// TIA Portal V16 export
// export: Created 2024-04-26T21:24:40.8001835Z, ExportSetting WithDefaults, DisplayName Totally Integrated Automation Portal, DisplayVersion V16, DisplayName TIA Portal Version Control Interface, DisplayVersion V16, DisplayName TIA Portal Openness, DisplayVersion V16, DisplayName STEP 7 Professional, DisplayVersion V16, DisplayName STEP 7 Safety, DisplayVersion V16, DisplayName WinCC Professional, DisplayVersion V16
ORGANIZATION_BLOCK "Main"   // OB1, LAD, ProgramCycle
TITLE = "Main Program Sweep (Cycle)"
{ S7_Optimized_Access := 'TRUE' }
VERSION : 0.1
// stored: AutoNumber true, IsIECCheckEnabled false, SetENOAutomatically false
   VAR_INPUT
      Initial_Call : Bool;   // Initial call of this OB
      Remanence : Bool;   // =True, if remanent data are available
   END_VAR
   VAR CONSTANT
      pozycja : Real := 45.0;
   END_VAR
   VAR_TEMP   // added for the SCL form of the ladder/FBD networks
      _w1 : Bool;
      _w2 : Bool;
   END_VAR
BEGIN

REGION Network 1: załączenie osi
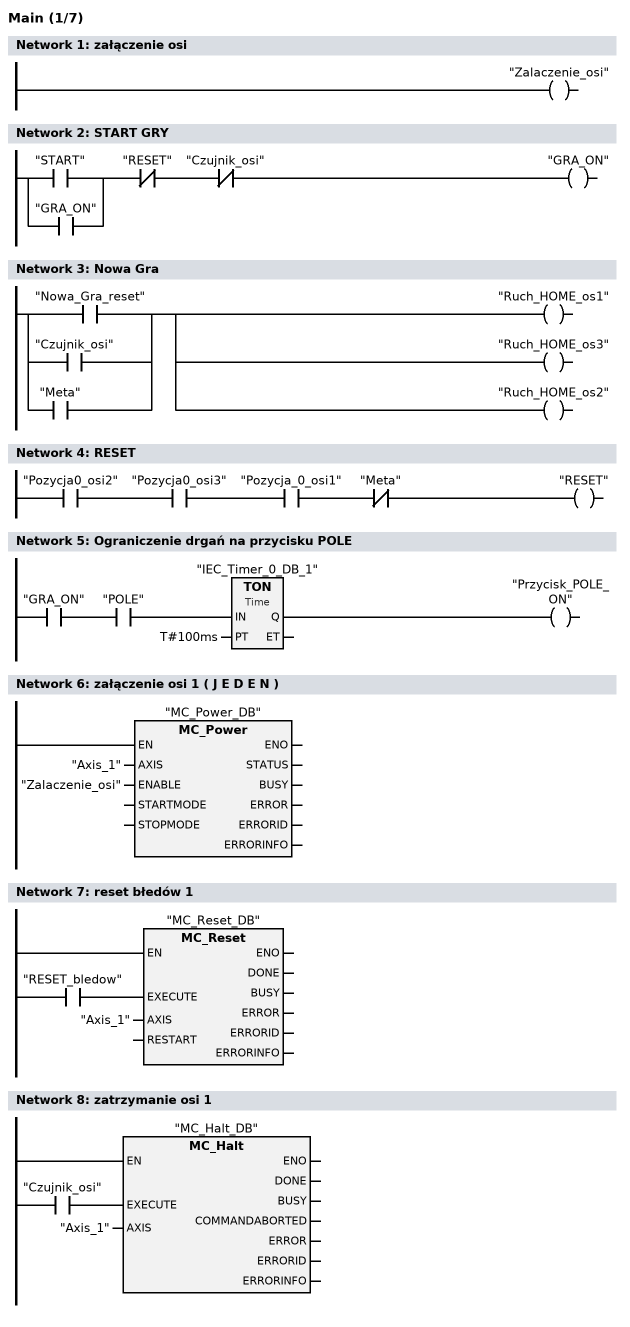
   RUNG wire#powerrail
      Coil( "Zalaczenie_osi" )
   END_RUNG
   // the same network as SCL:
   "Zalaczenie_osi" := TRUE;
END_REGION

REGION Network 2: START GRY
   RUNG wire#powerrail
      Contact( "START" )
      wire#w1
      I_Contact( "RESET" )
      I_Contact( "Czujnik_osi" )
      Coil( "GRA_ON" )
   END_RUNG
   RUNG wire#powerrail
      Contact( "GRA_ON" )
   END_RUNG wire#w1
   // the same network as SCL:
   "GRA_ON" := ("START" OR "GRA_ON") AND NOT "RESET" AND NOT "Czujnik_osi";
END_REGION

REGION Network 3: Nowa Gra
   RUNG wire#powerrail
      Contact( "Nowa_Gra_reset" )
      wire#w1
      Coil( "Ruch_HOME_os1" )
   END_RUNG
   RUNG wire#powerrail
      Contact( "Czujnik_osi" )
   END_RUNG wire#w1
   RUNG wire#powerrail
      Contact( "Meta" )
   END_RUNG wire#w1
   RUNG wire#w1
      Coil( "Ruch_HOME_os3" )
   END_RUNG
   RUNG wire#w1
      Coil( "Ruch_HOME_os2" )
   END_RUNG
   // the same network as SCL:
   "Ruch_HOME_os1" := "Nowa_Gra_reset" OR "Czujnik_osi" OR "Meta";
   "Ruch_HOME_os3" := "Ruch_HOME_os1";
   "Ruch_HOME_os2" := "Ruch_HOME_os1";
END_REGION

REGION Network 4: RESET
   RUNG wire#powerrail
      Contact( "Pozycja0_osi2" )
      Contact( "Pozycja0_osi3" )
      Contact( "Pozycja_0_osi1" )
      I_Contact( "Meta" )
      Coil( "RESET" )
   END_RUNG
   // the same network as SCL:
   "RESET" := "Pozycja0_osi2" AND "Pozycja0_osi3" AND "Pozycja_0_osi1" AND NOT "Meta";
END_REGION

REGION Network 5: Ograniczenie drgań na przycisku POLE
   RUNG wire#powerrail
      Contact( "GRA_ON" )
      Contact( "POLE" )
      { S7_Templates := "time_type := Time" } "IEC_Timer_0_DB_1".TON(pt := T#100ms, et =>)
      Coil( "Przycisk_POLE_ON" )
   END_RUNG
   // the same network as SCL:
   "IEC_Timer_0_DB_1".TON(IN := "GRA_ON" AND "POLE", PT := T#100ms);
   "Przycisk_POLE_ON" := "IEC_Timer_0_DB_1".Q;
END_REGION

REGION Network 6: załączenie osi 1 ( J E D E N )
   RUNG wire#powerrail
      "MC_Power_DB".MC_Power(Axis := "Axis_1", Enable := "Zalaczenie_osi", StartMode :=, StopMode :=, Status =>, Busy =>, Error =>, ErrorID =>, ErrorInfo =>)
   END_RUNG
   // the same network as SCL:
   "MC_Power_DB"(Axis := "Axis_1", Enable := "Zalaczenie_osi");   // MC_Power
END_REGION

REGION Network 7: reset błedów 1
   RUNG wire#powerrail
      "MC_Reset_DB".MC_Reset(Execute := wire#w1, Axis := "Axis_1", Restart :=, Done =>, Busy =>, Error =>, ErrorID =>, ErrorInfo =>)
   END_RUNG
   RUNG wire#powerrail
      Contact( "RESET_bledow" )
   END_RUNG wire#w1
   // the same network as SCL:
   "MC_Reset_DB"(Execute := "RESET_bledow", Axis := "Axis_1");   // MC_Reset
END_REGION

REGION Network 8: zatrzymanie osi 1
   RUNG wire#powerrail
      "MC_Halt_DB".MC_Halt(Execute := wire#w1, Axis := "Axis_1", Done =>, Busy =>, CommandAborted =>, Error =>, ErrorID =>, ErrorInfo =>)
   END_RUNG
   RUNG wire#powerrail
      Contact( "Czujnik_osi" )
   END_RUNG wire#w1
   // the same network as SCL:
   "MC_Halt_DB"(Execute := "Czujnik_osi", Axis := "Axis_1");   // MC_Halt
END_REGION

REGION Network 9: pozycjonowanie osi 1
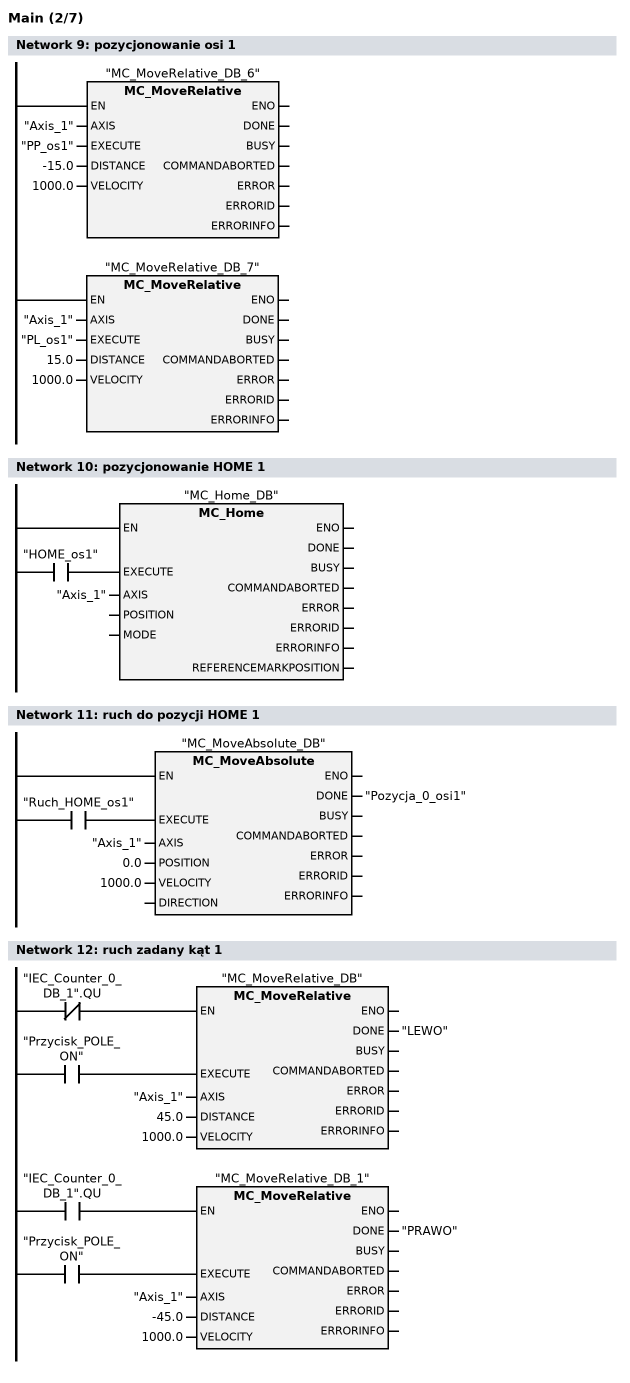
   RUNG wire#powerrail
      "MC_MoveRelative_DB_6".MC_MoveRelative(Axis := "Axis_1", Execute := "PP_os1", Distance := -15.0, Velocity := 1000.0, Done =>, Busy =>, CommandAborted =>, Error =>, ErrorID =>, ErrorInfo =>)
   END_RUNG
   RUNG wire#powerrail
      "MC_MoveRelative_DB_7".MC_MoveRelative(Axis := "Axis_1", Execute := "PL_os1", Distance := 15.0, Velocity := 1000.0, Done =>, Busy =>, CommandAborted =>, Error =>, ErrorID =>, ErrorInfo =>)
   END_RUNG
   // the same network as SCL:
   "MC_MoveRelative_DB_6"(Axis := "Axis_1", Execute := "PP_os1", Distance := -15.0, Velocity := 1000.0);   // MC_MoveRelative
   "MC_MoveRelative_DB_7"(Axis := "Axis_1", Execute := "PL_os1", Distance := 15.0, Velocity := 1000.0);   // MC_MoveRelative
END_REGION

REGION Network 10: pozycjonowanie HOME 1
   RUNG wire#powerrail
      "MC_Home_DB".MC_Home(Execute := wire#w1, Axis := "Axis_1", Position :=, Mode :=, Done =>, Busy =>, CommandAborted =>, Error =>, ErrorID =>, ErrorInfo =>, ReferenceMarkPosition =>)
   END_RUNG
   RUNG wire#powerrail
      Contact( "HOME_os1" )
   END_RUNG wire#w1
   // the same network as SCL:
   "MC_Home_DB"(Execute := "HOME_os1", Axis := "Axis_1");   // MC_Home
END_REGION

REGION Network 11: ruch do pozycji HOME 1
   RUNG wire#powerrail
      "MC_MoveAbsolute_DB".MC_MoveAbsolute(Execute := wire#w1, Axis := "Axis_1", Position := 0.0, Velocity := 1000.0, Direction :=, Done => "Pozycja_0_osi1", Busy =>, CommandAborted =>, Error =>, ErrorID =>, ErrorInfo =>)
   END_RUNG
   RUNG wire#powerrail
      Contact( "Ruch_HOME_os1" )
   END_RUNG wire#w1
   // the same network as SCL:
   "MC_MoveAbsolute_DB"(Execute := "Ruch_HOME_os1",   // MC_MoveAbsolute
                        Axis := "Axis_1",
                        Position := 0.0,
                        Velocity := 1000.0,
                        Done => "Pozycja_0_osi1");
END_REGION

REGION Network 12: ruch zadany kąt 1
   RUNG wire#powerrail
      I_Contact( "IEC_Counter_0_DB_1".QU )
      "MC_MoveRelative_DB".MC_MoveRelative(Execute := wire#w1, Axis := "Axis_1", Distance := 45.0, Velocity := 1000.0, Done => "LEWO", Busy =>, CommandAborted =>, Error =>, ErrorID =>, ErrorInfo =>)
   END_RUNG
   RUNG wire#powerrail
      Contact( "Przycisk_POLE_ON" )
   END_RUNG wire#w1
   RUNG wire#powerrail
      Contact( "IEC_Counter_0_DB_1".QU )
      "MC_MoveRelative_DB_1".MC_MoveRelative(Execute := wire#w2, Axis := "Axis_1", Distance := -45.0, Velocity := 1000.0, Done => "PRAWO", Busy =>, CommandAborted =>, Error =>, ErrorID =>, ErrorInfo =>)
   END_RUNG
   RUNG wire#powerrail
      Contact( "Przycisk_POLE_ON" )
   END_RUNG wire#w2
   // the same network as SCL:
   IF NOT "IEC_Counter_0_DB_1".QU THEN
       "MC_MoveRelative_DB"(Execute := "Przycisk_POLE_ON",   // MC_MoveRelative
                            Axis := "Axis_1",
                            Distance := 45.0,
                            Velocity := 1000.0,
                            Done => "LEWO");
   END_IF;
   IF "IEC_Counter_0_DB_1".QU THEN
       "MC_MoveRelative_DB_1"(Execute := "Przycisk_POLE_ON",   // MC_MoveRelative
                              Axis := "Axis_1",
                              Distance := -45.0,
                              Velocity := 1000.0,
                              Done => "PRAWO");
   END_IF;
END_REGION

REGION Network 13: Funkcja sekwencyjnego obracania 1
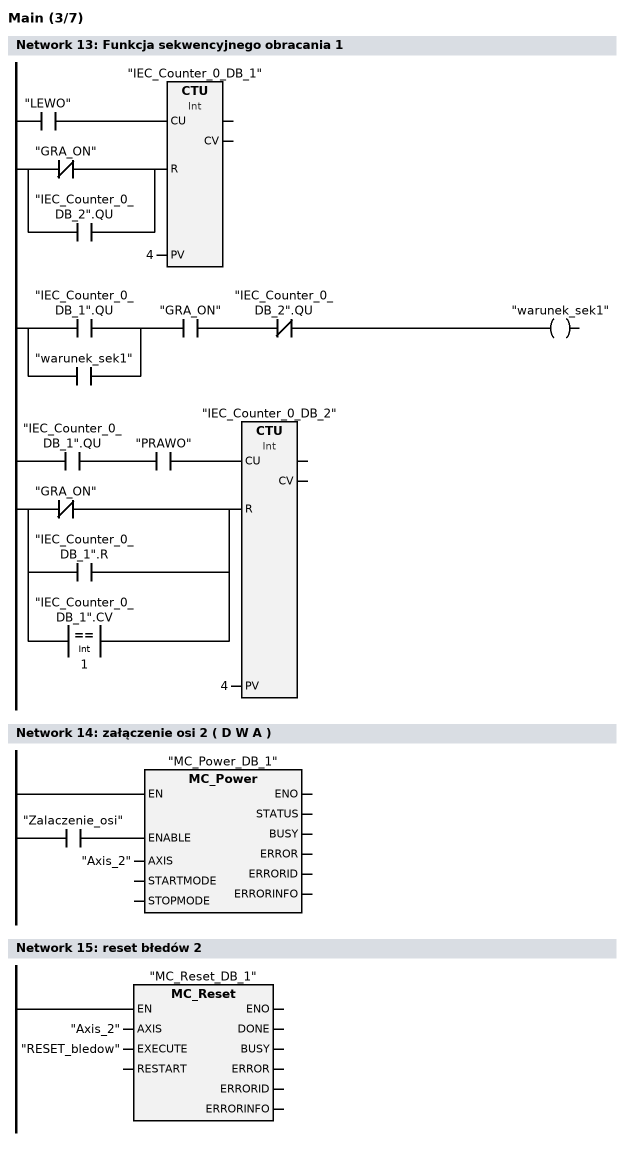
   RUNG wire#powerrail
      Contact( "LEWO" )
      { S7_Templates := "value_type := Int" } "IEC_Counter_0_DB_1".CTU(r := wire#w1, pv := 4, cv =>)
   END_RUNG
   RUNG wire#powerrail
      I_Contact( "GRA_ON" )
   END_RUNG wire#w1
   RUNG wire#powerrail
      Contact( "IEC_Counter_0_DB_2".QU )
   END_RUNG wire#w1
   RUNG wire#powerrail
      Contact( "IEC_Counter_0_DB_1".QU )
      wire#w2
      Contact( "GRA_ON" )
      I_Contact( "IEC_Counter_0_DB_2".QU )
      Coil( "warunek_sek1" )
   END_RUNG
   RUNG wire#powerrail
      Contact( "warunek_sek1" )
   END_RUNG wire#w2
   RUNG wire#powerrail
      Contact( "IEC_Counter_0_DB_1".QU )
      Contact( "PRAWO" )
      { S7_Templates := "value_type := Int" } "IEC_Counter_0_DB_2".CTU(r := wire#w3, pv := 4, cv =>)
   END_RUNG
   RUNG wire#powerrail
      I_Contact( "GRA_ON" )
   END_RUNG wire#w3
   RUNG wire#powerrail
      Contact( "IEC_Counter_0_DB_1".R )
   END_RUNG wire#w3
   RUNG wire#powerrail
      { S7_Templates := "SrcType := Int" } EQ_Contact(in1 := "IEC_Counter_0_DB_1".CV, in2 := 1)
   END_RUNG wire#w3
   // the same network as SCL:
   "IEC_Counter_0_DB_1".CTU(CU := "LEWO", R := NOT "GRA_ON" OR "IEC_Counter_0_DB_2".QU, PV := 4);
   "warunek_sek1" := ("IEC_Counter_0_DB_1".QU OR "warunek_sek1") AND "GRA_ON" AND NOT "IEC_Counter_0_DB_2".QU;
   "IEC_Counter_0_DB_2".CTU(CU := "IEC_Counter_0_DB_1".QU AND "PRAWO",
                           R := NOT "GRA_ON" OR "IEC_Counter_0_DB_1".R OR ("IEC_Counter_0_DB_1".CV = 1),
                           PV := 4);
END_REGION

REGION Network 14: załączenie osi 2 ( D W A )
   RUNG wire#powerrail
      "MC_Power_DB_1".MC_Power(Enable := wire#w1, Axis := "Axis_2", StartMode :=, StopMode :=, Status =>, Busy =>, Error =>, ErrorID =>, ErrorInfo =>)
   END_RUNG
   RUNG wire#powerrail
      Contact( "Zalaczenie_osi" )
   END_RUNG wire#w1
   // the same network as SCL:
   "MC_Power_DB_1"(Enable := "Zalaczenie_osi", Axis := "Axis_2");   // MC_Power
END_REGION

REGION Network 15: reset błedów 2
   RUNG wire#powerrail
      "MC_Reset_DB_1".MC_Reset(Axis := "Axis_2", Execute := "RESET_bledow", Restart :=, Done =>, Busy =>, Error =>, ErrorID =>, ErrorInfo =>)
   END_RUNG
   // the same network as SCL:
   "MC_Reset_DB_1"(Axis := "Axis_2", Execute := "RESET_bledow");   // MC_Reset
END_REGION

REGION Network 16: pozycjonowanie osi 2
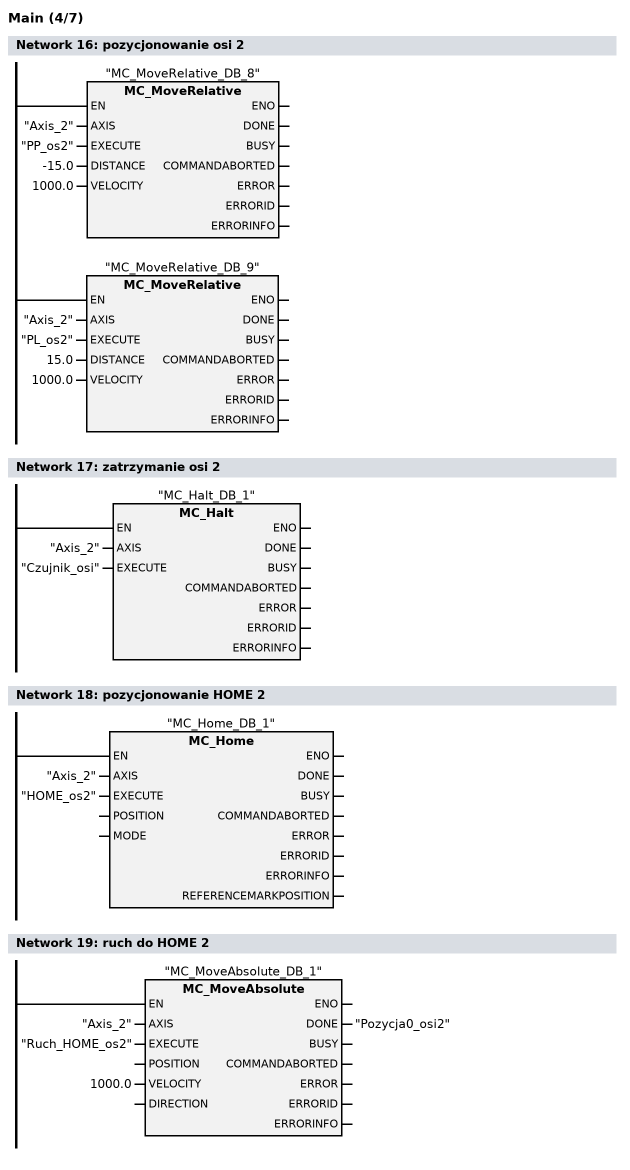
   RUNG wire#powerrail
      "MC_MoveRelative_DB_8".MC_MoveRelative(Axis := "Axis_2", Execute := "PP_os2", Distance := -15.0, Velocity := 1000.0, Done =>, Busy =>, CommandAborted =>, Error =>, ErrorID =>, ErrorInfo =>)
   END_RUNG
   RUNG wire#powerrail
      "MC_MoveRelative_DB_9".MC_MoveRelative(Axis := "Axis_2", Execute := "PL_os2", Distance := 15.0, Velocity := 1000.0, Done =>, Busy =>, CommandAborted =>, Error =>, ErrorID =>, ErrorInfo =>)
   END_RUNG
   // the same network as SCL:
   "MC_MoveRelative_DB_8"(Axis := "Axis_2", Execute := "PP_os2", Distance := -15.0, Velocity := 1000.0);   // MC_MoveRelative
   "MC_MoveRelative_DB_9"(Axis := "Axis_2", Execute := "PL_os2", Distance := 15.0, Velocity := 1000.0);   // MC_MoveRelative
END_REGION

REGION Network 17: zatrzymanie osi 2
   RUNG wire#powerrail
      "MC_Halt_DB_1".MC_Halt(Axis := "Axis_2", Execute := "Czujnik_osi", Done =>, Busy =>, CommandAborted =>, Error =>, ErrorID =>, ErrorInfo =>)
   END_RUNG
   // the same network as SCL:
   "MC_Halt_DB_1"(Axis := "Axis_2", Execute := "Czujnik_osi");   // MC_Halt
END_REGION

REGION Network 18: pozycjonowanie HOME 2
   RUNG wire#powerrail
      "MC_Home_DB_1".MC_Home(Axis := "Axis_2", Execute := "HOME_os2", Position :=, Mode :=, Done =>, Busy =>, CommandAborted =>, Error =>, ErrorID =>, ErrorInfo =>, ReferenceMarkPosition =>)
   END_RUNG
   // the same network as SCL:
   "MC_Home_DB_1"(Axis := "Axis_2", Execute := "HOME_os2");   // MC_Home
END_REGION

REGION Network 19: ruch do HOME 2
   RUNG wire#powerrail
      "MC_MoveAbsolute_DB_1".MC_MoveAbsolute(Axis := "Axis_2", Execute := "Ruch_HOME_os2", Position :=, Velocity := 1000.0, Direction :=, Done => "Pozycja0_osi2", Busy =>, CommandAborted =>, Error =>, ErrorID =>, ErrorInfo =>)
   END_RUNG
   // the same network as SCL:
   "MC_MoveAbsolute_DB_1"(Axis := "Axis_2",   // MC_MoveAbsolute
                          Execute := "Ruch_HOME_os2",
                          Velocity := 1000.0,
                          Done => "Pozycja0_osi2");
END_REGION

REGION Network 20: ruch zadany kąt 2
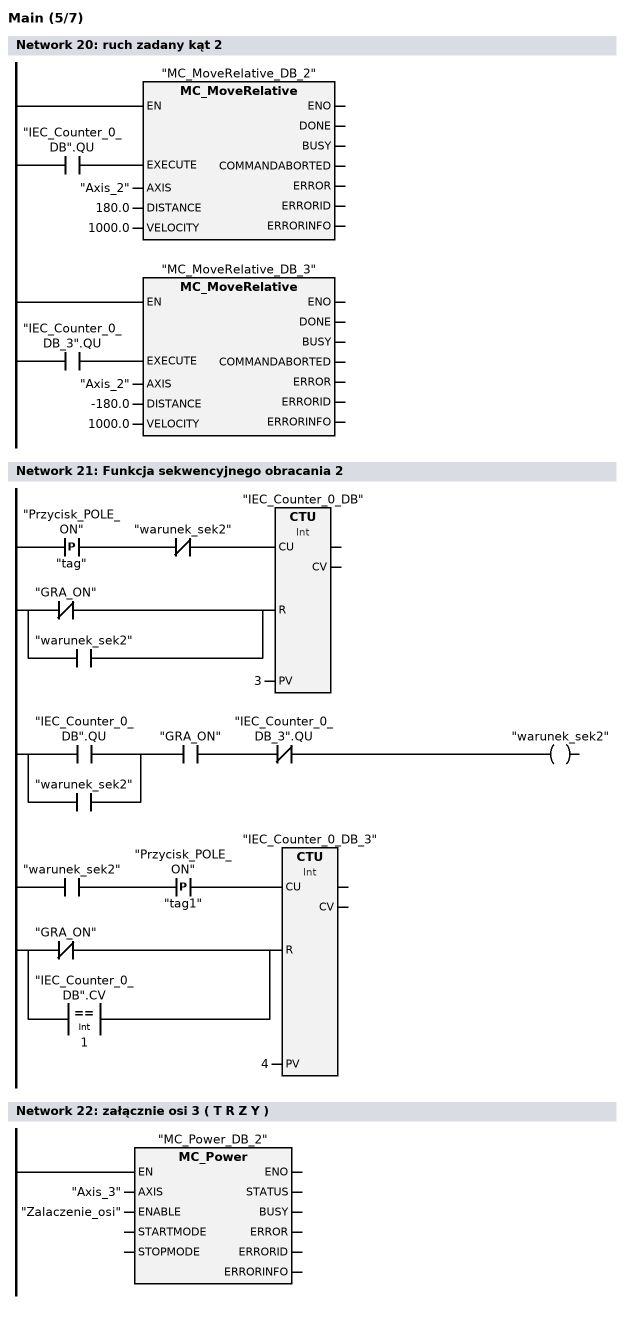
   RUNG wire#powerrail
      "MC_MoveRelative_DB_2".MC_MoveRelative(Execute := wire#w1, Axis := "Axis_2", Distance := 180.0, Velocity := 1000.0, Done =>, Busy =>, CommandAborted =>, Error =>, ErrorID =>, ErrorInfo =>)
   END_RUNG
   RUNG wire#powerrail
      Contact( "IEC_Counter_0_DB".QU )
   END_RUNG wire#w1
   RUNG wire#powerrail
      "MC_MoveRelative_DB_3".MC_MoveRelative(Execute := wire#w2, Axis := "Axis_2", Distance := -180.0, Velocity := 1000.0, Done =>, Busy =>, CommandAborted =>, Error =>, ErrorID =>, ErrorInfo =>)
   END_RUNG
   RUNG wire#powerrail
      Contact( "IEC_Counter_0_DB_3".QU )
   END_RUNG wire#w2
   // the same network as SCL:
   "MC_MoveRelative_DB_2"(Execute := "IEC_Counter_0_DB".QU,   // MC_MoveRelative
                          Axis := "Axis_2",
                          Distance := 180.0,
                          Velocity := 1000.0);
   "MC_MoveRelative_DB_3"(Execute := "IEC_Counter_0_DB_3".QU,   // MC_MoveRelative
                          Axis := "Axis_2",
                          Distance := -180.0,
                          Velocity := 1000.0);
END_REGION

REGION Network 21: Funkcja sekwencyjnego obracania 2
   RUNG wire#powerrail
      P_Contact(operand := "Przycisk_POLE_ON", bit := "tag")
      I_Contact( "warunek_sek2" )
      { S7_Templates := "value_type := Int" } "IEC_Counter_0_DB".CTU(r := wire#w1, pv := 3, cv =>)
   END_RUNG
   RUNG wire#powerrail
      I_Contact( "GRA_ON" )
   END_RUNG wire#w1
   RUNG wire#powerrail
      Contact( "warunek_sek2" )
   END_RUNG wire#w1
   RUNG wire#powerrail
      Contact( "IEC_Counter_0_DB".QU )
      wire#w2
      Contact( "GRA_ON" )
      I_Contact( "IEC_Counter_0_DB_3".QU )
      Coil( "warunek_sek2" )
   END_RUNG
   RUNG wire#powerrail
      Contact( "warunek_sek2" )
   END_RUNG wire#w2
   RUNG wire#powerrail
      Contact( "warunek_sek2" )
      P_Contact(operand := "Przycisk_POLE_ON", bit := "tag1")
      { S7_Templates := "value_type := Int" } "IEC_Counter_0_DB_3".CTU(r := wire#w3, pv := 4, cv =>)
   END_RUNG
   RUNG wire#powerrail
      I_Contact( "GRA_ON" )
   END_RUNG wire#w3
   RUNG wire#powerrail
      { S7_Templates := "SrcType := Int" } EQ_Contact(in1 := "IEC_Counter_0_DB".CV, in2 := 1)
   END_RUNG wire#w3
   // the same network as SCL:
   #_w1 := "Przycisk_POLE_ON" AND NOT "tag";   // rising edge of "Przycisk_POLE_ON"
   "tag" := "Przycisk_POLE_ON";
   "IEC_Counter_0_DB".CTU(CU := #_w1 AND NOT "warunek_sek2", R := NOT "GRA_ON" OR "warunek_sek2", PV := 3);
   "warunek_sek2" := ("IEC_Counter_0_DB".QU OR "warunek_sek2") AND "GRA_ON" AND NOT "IEC_Counter_0_DB_3".QU;
   #_w2 := "warunek_sek2" AND "Przycisk_POLE_ON" AND NOT "tag1";   // rising edge of "Przycisk_POLE_ON"
   "tag1" := "Przycisk_POLE_ON";
   "IEC_Counter_0_DB_3".CTU(CU := #_w2, R := NOT "GRA_ON" OR ("IEC_Counter_0_DB".CV = 1), PV := 4);
END_REGION

REGION Network 22: załącznie osi 3 ( T R Z Y )
   RUNG wire#powerrail
      "MC_Power_DB_2".MC_Power(Axis := "Axis_3", Enable := "Zalaczenie_osi", StartMode :=, StopMode :=, Status =>, Busy =>, Error =>, ErrorID =>, ErrorInfo =>)
   END_RUNG
   // the same network as SCL:
   "MC_Power_DB_2"(Axis := "Axis_3", Enable := "Zalaczenie_osi");   // MC_Power
END_REGION

REGION Network 23: reset błądów osi 3
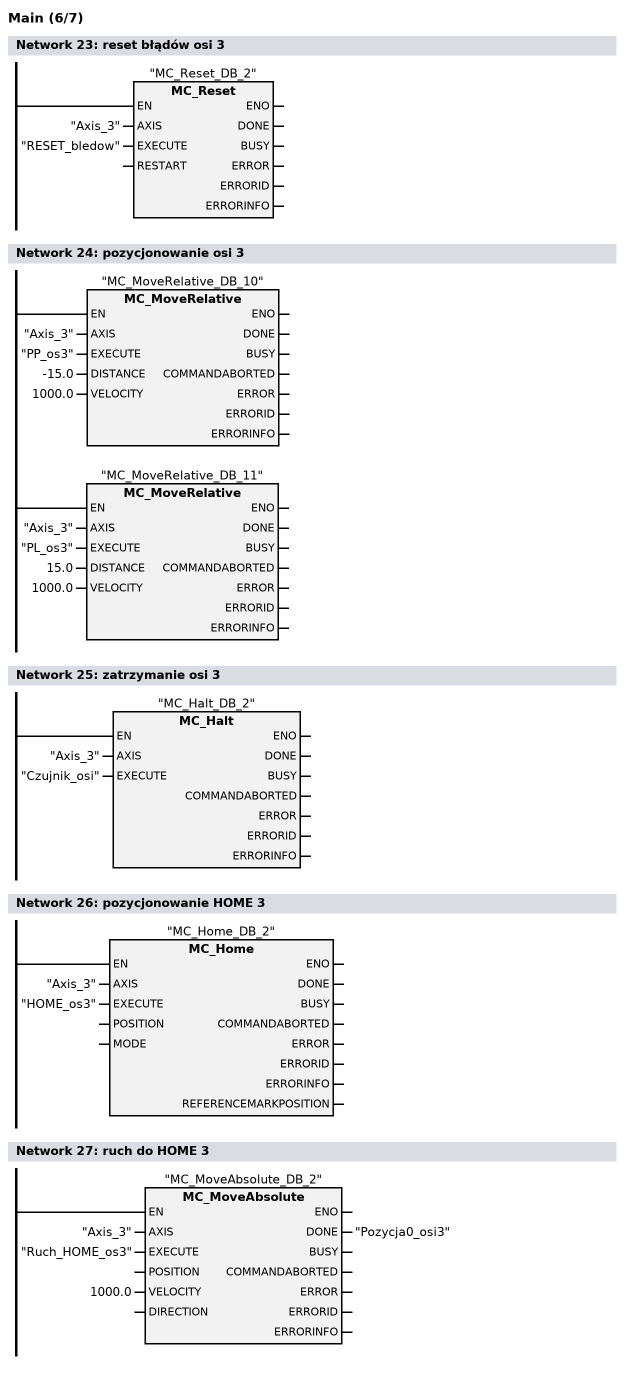
   RUNG wire#powerrail
      "MC_Reset_DB_2".MC_Reset(Axis := "Axis_3", Execute := "RESET_bledow", Restart :=, Done =>, Busy =>, Error =>, ErrorID =>, ErrorInfo =>)
   END_RUNG
   // the same network as SCL:
   "MC_Reset_DB_2"(Axis := "Axis_3", Execute := "RESET_bledow");   // MC_Reset
END_REGION

REGION Network 24: pozycjonowanie osi 3
   RUNG wire#powerrail
      "MC_MoveRelative_DB_10".MC_MoveRelative(Axis := "Axis_3", Execute := "PP_os3", Distance := -15.0, Velocity := 1000.0, Done =>, Busy =>, CommandAborted =>, Error =>, ErrorID =>, ErrorInfo =>)
   END_RUNG
   RUNG wire#powerrail
      "MC_MoveRelative_DB_11".MC_MoveRelative(Axis := "Axis_3", Execute := "PL_os3", Distance := 15.0, Velocity := 1000.0, Done =>, Busy =>, CommandAborted =>, Error =>, ErrorID =>, ErrorInfo =>)
   END_RUNG
   // the same network as SCL:
   "MC_MoveRelative_DB_10"(Axis := "Axis_3", Execute := "PP_os3", Distance := -15.0, Velocity := 1000.0);   // MC_MoveRelative
   "MC_MoveRelative_DB_11"(Axis := "Axis_3", Execute := "PL_os3", Distance := 15.0, Velocity := 1000.0);   // MC_MoveRelative
END_REGION

REGION Network 25: zatrzymanie osi 3
   RUNG wire#powerrail
      "MC_Halt_DB_2".MC_Halt(Axis := "Axis_3", Execute := "Czujnik_osi", Done =>, Busy =>, CommandAborted =>, Error =>, ErrorID =>, ErrorInfo =>)
   END_RUNG
   // the same network as SCL:
   "MC_Halt_DB_2"(Axis := "Axis_3", Execute := "Czujnik_osi");   // MC_Halt
END_REGION

REGION Network 26: pozycjonowanie HOME 3
   RUNG wire#powerrail
      "MC_Home_DB_2".MC_Home(Axis := "Axis_3", Execute := "HOME_os3", Position :=, Mode :=, Done =>, Busy =>, CommandAborted =>, Error =>, ErrorID =>, ErrorInfo =>, ReferenceMarkPosition =>)
   END_RUNG
   // the same network as SCL:
   "MC_Home_DB_2"(Axis := "Axis_3", Execute := "HOME_os3");   // MC_Home
END_REGION

REGION Network 27: ruch do HOME 3
   RUNG wire#powerrail
      "MC_MoveAbsolute_DB_2".MC_MoveAbsolute(Axis := "Axis_3", Execute := "Ruch_HOME_os3", Position :=, Velocity := 1000.0, Direction :=, Done => "Pozycja0_osi3", Busy =>, CommandAborted =>, Error =>, ErrorID =>, ErrorInfo =>)
   END_RUNG
   // the same network as SCL:
   "MC_MoveAbsolute_DB_2"(Axis := "Axis_3",   // MC_MoveAbsolute
                          Execute := "Ruch_HOME_os3",
                          Velocity := 1000.0,
                          Done => "Pozycja0_osi3");
END_REGION

REGION Network 28: ruch o zadany kąt 3
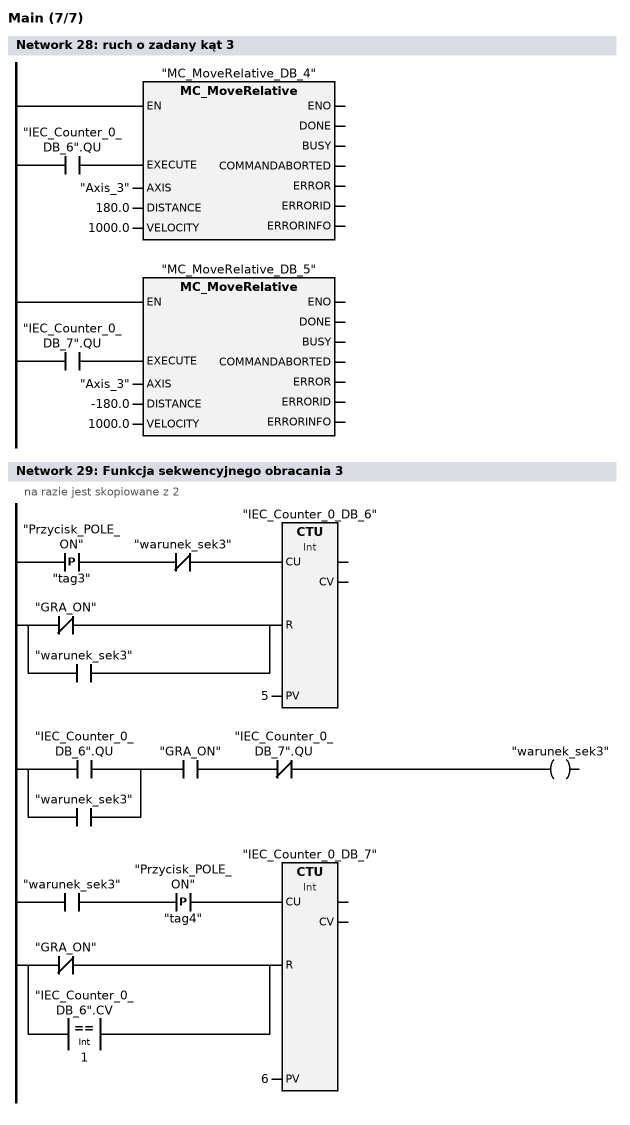
   RUNG wire#powerrail
      "MC_MoveRelative_DB_4".MC_MoveRelative(Execute := wire#w1, Axis := "Axis_3", Distance := 180.0, Velocity := 1000.0, Done =>, Busy =>, CommandAborted =>, Error =>, ErrorID =>, ErrorInfo =>)
   END_RUNG
   RUNG wire#powerrail
      Contact( "IEC_Counter_0_DB_6".QU )
   END_RUNG wire#w1
   RUNG wire#powerrail
      "MC_MoveRelative_DB_5".MC_MoveRelative(Execute := wire#w2, Axis := "Axis_3", Distance := -180.0, Velocity := 1000.0, Done =>, Busy =>, CommandAborted =>, Error =>, ErrorID =>, ErrorInfo =>)
   END_RUNG
   RUNG wire#powerrail
      Contact( "IEC_Counter_0_DB_7".QU )
   END_RUNG wire#w2
   // the same network as SCL:
   "MC_MoveRelative_DB_4"(Execute := "IEC_Counter_0_DB_6".QU,   // MC_MoveRelative
                          Axis := "Axis_3",
                          Distance := 180.0,
                          Velocity := 1000.0);
   "MC_MoveRelative_DB_5"(Execute := "IEC_Counter_0_DB_7".QU,   // MC_MoveRelative
                          Axis := "Axis_3",
                          Distance := -180.0,
                          Velocity := 1000.0);
END_REGION

REGION Network 29: Funkcja sekwencyjnego obracania 3
   // na razie jest skopiowane z 2
   RUNG wire#powerrail
      P_Contact(operand := "Przycisk_POLE_ON", bit := "tag3")
      I_Contact( "warunek_sek3" )
      { S7_Templates := "value_type := Int" } "IEC_Counter_0_DB_6".CTU(r := wire#w1, pv := 5, cv =>)
   END_RUNG
   RUNG wire#powerrail
      I_Contact( "GRA_ON" )
   END_RUNG wire#w1
   RUNG wire#powerrail
      Contact( "warunek_sek3" )
   END_RUNG wire#w1
   RUNG wire#powerrail
      Contact( "IEC_Counter_0_DB_6".QU )
      wire#w2
      Contact( "GRA_ON" )
      I_Contact( "IEC_Counter_0_DB_7".QU )
      Coil( "warunek_sek3" )
   END_RUNG
   RUNG wire#powerrail
      Contact( "warunek_sek3" )
   END_RUNG wire#w2
   RUNG wire#powerrail
      Contact( "warunek_sek3" )
      P_Contact(operand := "Przycisk_POLE_ON", bit := "tag4")
      { S7_Templates := "value_type := Int" } "IEC_Counter_0_DB_7".CTU(r := wire#w3, pv := 6, cv =>)
   END_RUNG
   RUNG wire#powerrail
      I_Contact( "GRA_ON" )
   END_RUNG wire#w3
   RUNG wire#powerrail
      { S7_Templates := "SrcType := Int" } EQ_Contact(in1 := "IEC_Counter_0_DB_6".CV, in2 := 1)
   END_RUNG wire#w3
   // the same network as SCL:
   #_w1 := "Przycisk_POLE_ON" AND NOT "tag3";   // rising edge of "Przycisk_POLE_ON"
   "tag3" := "Przycisk_POLE_ON";
   "IEC_Counter_0_DB_6".CTU(CU := #_w1 AND NOT "warunek_sek3", R := NOT "GRA_ON" OR "warunek_sek3", PV := 5);
   "warunek_sek3" := ("IEC_Counter_0_DB_6".QU OR "warunek_sek3") AND "GRA_ON" AND NOT "IEC_Counter_0_DB_7".QU;
   #_w2 := "warunek_sek3" AND "Przycisk_POLE_ON" AND NOT "tag4";   // rising edge of "Przycisk_POLE_ON"
   "tag4" := "Przycisk_POLE_ON";
   "IEC_Counter_0_DB_7".CTU(CU := #_w2, R := NOT "GRA_ON" OR ("IEC_Counter_0_DB_6".CV = 1), PV := 6);
END_REGION
END_ORGANIZATION_BLOCK
